{attribute addProperty BoxType "ATH2040-5250-0022"}
{attribute addProperty Id "BinaryDataAT %I*ARRAY [0..59] OF BYTE00"}
{attribute addProperty CRC "385037607"}
{attribute addProperty SizeInBites "0"}
{attribute addProperty SizeInBytes "0"}
TYPE FB_Inputs_16F33527 :
STRUCT
	{attribute addProperty Name "BinaryData"}
	BinaryData AT %I* : ARRAY [0..59] OF BYTE;
END_STRUCT
END_TYPE

(* stored: Version 1.2.0.0, ProductVersion 3.1.4024.9
   DUT FB_Inputs_16F33527: Id {d7a26ced-a7d0-4b98-b9db-a11fb1c55900} *)
